TYPE ST_Safety_ContactorEDM :
STRUCT
	b_MccbMasterEDM						: BOOL;
	b_MccbSlaveEDM						: BOOL;
	b_NetcontactorEDM					: BOOL;
	b_DcMccbEDM							: BOOL;
END_STRUCT
END_TYPE

(* stored: Version 1.1.0.1, ProductVersion 3.1.4026.18
   DUT ST_Safety_ContactorEDM: Id {c197fa78-a5d0-4337-b3fe-1db495539126} *)
